{attribute 'GeneratedUsingTerminal: EK1100-0000-0018'}
{attribute addProperty BoxType "EK1100-0000-0018"}
{attribute addProperty Id "Beckhoff_EJ9xxxEK1122Beckhoff_EJ9xxxEK1122_263487052A_0001_EJ9001_0000_0016EJ9001_AB5A94672A_0002_EJ9505_0000_0016EJ9505_B1D2CB3F6A_0003_EJ9576_0000_0018EJ9576_6F5CE42328A_0004_EJ9576_0000_0019EJ9576_8784E5ED29A_0005_EJ9576_0000_0020EJ9576_1238494C28A_0006_EJ9576_0000_0022EJ9576_C60EFF2F29"}
{attribute addProperty CRC "4149172018"}
{attribute addProperty Size "124"}
TYPE Beckhoff_EJ9xxx_F74F5732 EXTENDS EK1100_AB5A9467 :
STRUCT
	{attribute addProperty Name "Beckhoff_EJ9xxxEK1122"}
	{attribute addProperty PreviousPort "Beckhoff EJ9xxx : B"}
	Beckhoff_EJ9xxxEK1122 : Beckhoff_EJ9xxxEK1122_26348705;
	{attribute addProperty Name "A_0001_EJ9001_0000_0016"}
	{attribute addProperty PreviousPort "Beckhoff EJ9xxxEK1122 : C"}
	A_0001_EJ9001_0000_0016 : EJ9001_AB5A9467;
	{attribute addProperty Name "A_0002_EJ9505_0000_0016"}
	{attribute addProperty PreviousPort "A_0001(EJ9001-0000-0016) : B"}
	A_0002_EJ9505_0000_0016 : EJ9505_B1D2CB3F;
	{attribute addProperty Name "A_0003_EJ9576_0000_0018"}
	{attribute addProperty PreviousPort "A_0002(EJ9505-0000-0016) : B"}
	A_0003_EJ9576_0000_0018 : EJ9576_6F5CE423;
	{attribute addProperty Name "A_0004_EJ9576_0000_0019"}
	{attribute addProperty PreviousPort "A_0003(EJ9576-0000-0018) : B"}
	A_0004_EJ9576_0000_0019 : EJ9576_8784E5ED;
	{attribute addProperty Name "A_0005_EJ9576_0000_0020"}
	{attribute addProperty PreviousPort "A_0004(EJ9576-0000-0019) : B"}
	A_0005_EJ9576_0000_0020 : EJ9576_1238494C;
	{attribute addProperty Name "A_0006_EJ9576_0000_0022"}
	{attribute addProperty PreviousPort "A_0005(EJ9576-0000-0020) : B"}
	A_0006_EJ9576_0000_0022 : EJ9576_C60EFF2F;
END_STRUCT
END_TYPE

(* stored: Version 1.2.0.0, ProductVersion 3.1.4024.9
   DUT Beckhoff_EJ9xxx_F74F5732: Id {87d437d2-4f55-4ca3-b9ec-5d852b91a7c7} *)
